// SIMATIC S7-200 project (STEP 7-Micro/WIN), CPU 226 REL 01.23

SYMBOL_TABLE analog & its vd
oil_pipe_temp0   AIW0     // oil pipe temperature channel
oil_tank_temp0   AIW2     // oil tank temperature channel
motor_draft_temp0 AIW4     // motor draft temperature channel
motor_coil1_temp0 AIW6     // motor coil 1 temperature channel
motor_coil2_temp0 AIW8     // motor coil 2 temperature channel
motor_coil3_temp0 AIW10    // motor coil 3 temperature channel
fou_out_temp0    AIW12    // fourth stage out temperature channel
thi_out_temp0    AIW14    // third stage out temperature channel
sec_out_temp0    AIW16    // second stage out temperature channel
fir_out_temp0    AIW18    // first stage out temperature channel
oil_pre0         AIW20    // oil pressure channel
delivery_pre0    AIW22    // delivery pressure channel
fou_out_pre0     AIW24    // 4th stage  out pressure channel
thi_out_pre0     AIW26    // 3rd stage  out pressure channel
sec_out_pre0     AIW28    // 2nd stage  out pressure channel
fir_out_pre0     AIW30    // 1st stage  out pressure channel
fir_in_pre0      AIW32    // 1st stage  in pressure channel
oil_pipe_temp1   VD200    // oil pipe temperature value
oil_tank_temp1   VD204    // oil tank temperature value
motor_draft_temp1 VD208    // motor draft temperature value
motor_coil3_temp1 VD212    // motor coil 1 temperature value
motor_coil2_temp1 VD216    // motor coil 2 temperature value
motor_coil1_temp1 VD220    // motor coil 3 temperature value
fou_out_temp1    VD224    // fourth stage out temperature value
thi_out_temp1    VD228    // third stage out temperature value
sec_out_temp1    VD232    // second stage out temperature value
fir_out_temp1    VD236    // first stage out temperature value
oil_pre1         VD240    // oil pressure value
delivery_pre1    VD244    // delivery pressure value
fou_out_pre1     VD248    // 4th stage  out pressure value
thi_out_pre1     VD252    // 3rd stage  out pressure value
sec_out_pre1     VD256    // 2nd stage  out pressure value
fir_out_pre1     VD260    // 1st stage  out pressure value
fir_in_pre1      VD264    // 1st stage  in pressure value
END_SYMBOL_TABLE

SYMBOL_TABLE define_m
fou_out_p_hi_p_m M10.0
oil_p_low_p_m    M10.1
fir_o_t_hi_p_m   M10.2
sec_o_t_hi_p_m   M10.3
thi_o_t_hi_p_m   M10.4
fou_o_t_hi_p_m   M10.5
fir_coil_t_hi_p_m M10.6
sec_coil_t_hi_p_m M10.7
thi_coil_t_hi_p_m M11.0
draft_t_hi_p_m   M11.1
oil_t_hi_p_m     M11.2
fir_in_p_low_p_m M11.3
fir_in_p_hi_p_m  M11.4
delivery_p_hi_p_m M11.5
fou_o_p_hi_a_m   M14.0
oil_p_low_a_m    M14.1
fir_o_t_hi_a_m   M14.2
sec_o_t_hi_a_m   M14.3
thi_o_t_hi_a_m   M14.4
fou_o_t_hi_a_m   M14.5
fir_coil_t_hi_a_m M14.6
sec_coil_t_hi_a_m M14.7
thi_coil_t_hi_a_m M15.0
draft_t_hi_a_m   M15.1
oil_t_hi_a_m     M15.2
fir_in_p_low_a_m M15.3
fir_in_p_hi_a_m  M15.4
delivery_p_hi_a_m M15.5
oil_start_heat_m M15.6
oil_stop_heat_m  M15.7
sec_pre_high_m   M16.0
thi_pre_high_m   M16.1
fou_pre_high_m   M16.2
a_cooling_fan    M19.0
a_aid_pump       M19.1
a_infuse_pump    M19.2
a_water_pump     M19.3
a_main_motor     M19.5
m_main_start     M25.0
m_main_stop      M25.1
m_cooling_fan    M25.2
m_venting_fan    M25.3
m_infuse_pump    M25.4
m_oil_heater     M25.5
m_oil_pump       M25.6
m_water_pump     M25.7
m_fir_vavle      M26.0
m_sec_vavle      M26.1
m_thi_vavle      M26.2
m_fou_vavle      M26.3
a_pro_unlock     M7.0
fou_o_p_hi_unlock M7.1
oil_p_low_unlock M7.2
fir_o_t_hi_unlock M7.3
sec_o_t_hi_unlock M7.4
thi_o_t_hi_unlock M7.5
fou_o_t_hi_unlock M7.6
fir_coil_t_hi_unlock M7.7
sec_coil_t_hi_unlock M8.0
thi_coil_t_hi_unlock M8.1
draft_t_hi_unlock M8.2
oil_t_hi_unlock  M8.3
fir_in_p_low_unlock M8.4
fir_in_p_hi_unlock M8.5
delivery_p_hi_unlock M8.6
END_SYMBOL_TABLE

SYMBOL_TABLE pro & ala setting
fou_o_p_hi_p_s   VD300    // 4th stage out pressure high protect
oil_p_low_p_s    VD304    // oilt pressure low protect
fir_o_t_hi_p_s   VD308    // 1st stage out temperature high protect
sec_o_t_hi_p_s   VD312    // 2nd stage out temperature high protect
thi_o_t_hi_p_s   VD316    // 3rd stage out temperature high protect
fou_o_t_hi_p_s   VD320    // 4th stage out temperature high protect
fir_coil_t_hi_p_s VD324    // 1st coil temperature high protect
sec_coil_t_hi_p_s VD328    // 2nd coil temperature high protect
thi_coil_t_hi_p_s VD332    // 3rd coil out temperature high protect
draft_t_hi_p_s   VD336    // draft temperature high protect
oil_t_hi_p_s     VD340    // oil temperature high protect
fir_in_p_low_p_s VD344    // 1st stage in pressure low protect
fir_in_p_hi_p_s  VD348    // 1st stage in pressure high protect
delivery_p_hi_p_s VD352    // delivery pressure high protect
fou_o_p_hi_a_s   VD400    // 4th stage out pressure high alarm
oil_p_low_a_s    VD404    // oilt pressure low alarm
fir_o_t_hi_a_s   VD408    // 1st stage out temperature high alarm
sec_o_t_hi_a_s   VD412    // 2nd stage out temperature high alarm
thi_o_t_hi_a_s   VD416    // 3rd stage out temperature high alarm
fou_o_t_hi_a_s   VD420    // 4th stage out temperature high alarm
fir_coil_t_hi_a_s VD424    // 1st coil temperature high alarm
sec_coil_t_hi_a_s VD428    // 2nd coil temperature high alarm
thi_coil_t_hi_a_s VD432    // 3rd coil out temperature high alarm
draft_t_hi_a_s   VD436    // draft temperature high alarm
oil_t_hi_a_s     VD440    // oil temperature high alarm
fir_in_p_low_a_s VD444    // 1st stage in pressure low alarm
fir_in_p_hi_a_s  VD448    // 1st stage in pressure high alarm
delivery_p_hi_a_s VD452    // delivery pressure high alarm
oil_start_heat_s VD456    // temperature that oil start to heat
oil_stop_heat_s  VD460    // temperature that oil stop to heat
sec_pre_hi_s     VD464    // second stage out  pressure high alarm
thi_pre_hi_s     VD468    // third stage out  pressure high alarm
fou_pre_hi_s     VD472    // fourth stage out  pressure high alarm
invalid_time     VW490    // unvalid running time
fan_stop_time    VW492    // time when relay to stop fan
next_start_time  VW494    // interval when run again
test_oil_time    VW496    // time when relay to test oil pressure
fir_in_p_test_time VW498    // time to relay to test first stage input pressure
stop_aid_pump_time VW500    // time relay to stop the aid oil pump when main motor start
vavle_relay_time VW502    // time relay to open vavle  when main motor start
interval_time    VW504    // when start automatically ,the interval to start step by step
main_relay_time  VW506    // after all aid equipment running,to start main motor time
relay_stop_water VW508    // when stop system ,relay time to stop water pump
relay_stop_oil   VW510    // when stop system ,relay time to stop oil pump
relay_to_test_fir_pre VW512    // when 3# vavle is open  ,relay time to test inlet pressure
END_SYMBOL_TABLE

SYMBOL_TABLE i/o
main_motor_run   I0.0
main_motor_fault I0.1
cooling_fan_run  I0.2
cooling_fan_fault I0.3
vent_fan_run     I0.4
vent_fan_fault   I0.5
infuse_oil_pump_run I0.6
infuse_oil_pump_fault I0.7
heater_run       I1.0
heater_fault     I1.1
fir_vavle_open   I1.2
sec_vavle_open   I1.3
thi_vavle_open   I1.4
esd              I1.5
local_remote     I1.6
automatic        I1.7
manu             I2.0
gas_leakage      I2.1
test             I2.2
confirm          I2.3
reset            I2.4
start_button     I2.5
stop_button      I2.6
spare            I2.7
main_motor_start Q0.0
main_motor_stop  Q0.1
cooling_fan_st   Q0.2
venting_fan_st   Q0.3
infuse_oil_pump_st Q0.4
oil_heater_st    Q0.5
oil_pump_st      Q0.6
water_pump_st    Q0.7
fir_vavle_st     Q1.0
sec_vavle_st     Q1.1
thi_vavle_st     Q1.2
fou_vavle_st     Q1.3
spare_q_2        Q1.4
est_output       Q1.5
permit_indicator Q1.6
alarm_out        Q1.7
END_SYMBOL_TABLE

ORGANIZATION_BLOCK MAIN:OB1
TITLE=“CNG加气站控制程序”。
// 
// 系统中，四级出口压力超过四级出口压力高保护设定值且四级出口压力高保护解除标志  未置位时，必须触发 四级出口压力高保护标志，以防止压缩机因压力过高受损；
// 同样，当 油压低于 油压低保护设定值且主电机运行 时，必须触发 油压低保护标志，确保润滑系统正常。
// 
// 自动控制 模块按照预定顺序启动设备：首先激活 冷却风扇自动控制标志，通过 启动延时定时器 延时后启动 辅助泵自动控制标志，依次启动 输油泵自动控制标志、水泵自动控制标志，最后启动 主电机自动控制标志，每步之间必须有延时以确保设备稳定运行。
// 输出控制 根据逻辑驱动实际设备，主电机启动输出 仅在 主电机自动控制标志或手动启动信号有效时才能置位，而 报警输出 必须在系统异常（如 四级出口压力高保护标志 触发时）或紧急停机触发时激活，确保操作员及时响应。
// 
// 报警逻辑监测异常情况，当 四级出口压力超过 四级出口压力高报警设定值 时，必须触发 四级出口压力高报警标志，提醒维护人员检查系统。
// 此外，恢复出厂设置功能允许将 四级出口压力高保护设定值等参数重置为默认值（25.0）。
BEGIN
Network 1 // 网络标题
// 网络注释
LD     SM0.0
LPS
CALL   analog:SBR0
AN     a_pro_unlock:M7.0
CALL   protect:SBR1
LRD
CALL   alarm:SBR6
LPP
AW=    0, MW10
=      M28.0
Network 2 // 网络标题
// 网络注释
LDN    automatic:I1.7
AN     manu:I2.0
=      M28.5
Network 3
LD     reset:I2.4
MOVW   0, MW10
MOVW   0, MW14
MOVW   0, MW16
Network 4
LDN    main_motor_fault:I0.1
AN     cooling_fan_fault:I0.3
AN     vent_fan_fault:I0.5
AN     infuse_oil_pump_fault:I0.7
AN     heater_fault:I1.1
=      M28.1
Network 5
LD     M28.0
A      M28.1
AN     esd:I1.5
A      automatic:I1.7
CALL   auto:SBR2
Network 6
LDN    M28.0
ON     M28.1
O      esd:I1.5
ON     automatic:I1.7
MOVW   0, MW19
=      alarm_out:Q1.7
Network 7
LDN    manu:I2.0
MOVW   0, MW25
Network 8
LD     confirm:I2.3
A      reset:I2.4
TON    T40, 100
Network 9
LD     T40
CALL   recovery:SBR7
Network 10
LD     automatic:I1.7
O      manu:I2.0
A      M28.0
A      M28.1
AN     esd:I1.5
AN     M0.0
CALL   out:SBR4
Network 11 // 网络标题
// 网络注释
LD     esd:I1.5
=      est_output:Q1.5
END_ORGANIZATION_BLOCK

SUBROUTINE_BLOCK analog:SBR0
TITLE=子程序注释
BEGIN
Network 1
LD     SM0.0
CALL   Temperature:SBR11, oil_pipe_temp0:AIW0, oil_pipe_temp1:VD200
CALL   Temperature:SBR11, oil_tank_temp0:AIW2, oil_tank_temp1:VD204
CALL   Temperature:SBR11, motor_draft_temp0:AIW4, motor_draft_temp1:VD208
CALL   Temperature:SBR11, motor_coil3_temp0:AIW10, motor_coil3_temp1:VD212
CALL   Temperature:SBR11, motor_coil2_temp0:AIW8, motor_coil2_temp1:VD216
CALL   Temperature:SBR11, motor_coil1_temp0:AIW6, motor_coil1_temp1:VD220
CALL   Temperature:SBR11, fou_out_temp0:AIW12, fou_out_temp1:VD224
CALL   Temperature:SBR11, thi_out_temp0:AIW14, thi_out_temp1:VD228
CALL   Temperature:SBR11, sec_out_temp0:AIW16, sec_out_temp1:VD232
CALL   Temperature:SBR11, fir_out_temp0:AIW18, fir_out_temp1:VD236
Network 2 // 网络标题
// 网络注释
LD     SM0.0
CALL   Pressure:SBR12, oil_pre0:AIW20, 1.6, oil_pre1:VD240
CALL   Pressure:SBR12, delivery_pre0:AIW22, 40.0, delivery_pre1:VD244
CALL   Pressure:SBR12, fou_out_pre0:AIW24, 40.0, fou_out_pre1:VD248
CALL   Pressure:SBR12, thi_out_pre0:AIW26, 25.0, thi_out_pre1:VD252
CALL   Pressure:SBR12, sec_out_pre0:AIW28, 10.0, sec_out_pre1:VD256
CALL   Pressure:SBR12, fir_out_pre0:AIW30, 4.0, fir_out_pre1:VD260
CALL   Pressure:SBR12, fir_in_pre0:AIW32, 1.6, fir_in_pre1:VD264
END_SUBROUTINE_BLOCK

SUBROUTINE_BLOCK protect:SBR1
TITLE=
BEGIN
Network 1
LDR>=  fou_out_pre1:VD248, fou_o_p_hi_p_s:VD300
O      fou_out_p_hi_p_m:M10.0
AN     fou_o_p_hi_unlock:M7.1
=      fou_out_p_hi_p_m:M10.0
Network 2
LD     oil_pump_st:Q0.6
TON    T38, test_oil_time:VW496
Network 3
LD     T38
O      M19.6
AR>=   oil_p_low_p_s:VD304, oil_pre1:VD240
O      oil_p_low_p_m:M10.1
AN     oil_p_low_unlock:M7.2
=      oil_p_low_p_m:M10.1
Network 4
LDR>=  fir_out_temp1:VD236, fir_o_t_hi_p_s:VD308
O      fir_o_t_hi_p_m:M10.2
AN     fir_o_t_hi_unlock:M7.3
=      fir_o_t_hi_p_m:M10.2
Network 5
LDR>=  sec_out_temp1:VD232, sec_o_t_hi_p_s:VD312
O      sec_o_t_hi_p_m:M10.3
AN     sec_o_t_hi_unlock:M7.4
=      sec_o_t_hi_p_m:M10.3
Network 6
LDR>=  thi_out_temp1:VD228, thi_o_t_hi_p_s:VD316
O      thi_o_t_hi_p_m:M10.4
AN     thi_o_t_hi_unlock:M7.5
=      thi_o_t_hi_p_m:M10.4
Network 7
LDR>=  fou_out_temp1:VD224, fou_o_t_hi_p_s:VD320
O      fou_o_t_hi_p_m:M10.5
AN     fou_o_t_hi_unlock:M7.6
=      fou_o_t_hi_p_m:M10.5
Network 8
LDR>=  motor_coil1_temp1:VD220, fir_coil_t_hi_p_s:VD324
O      fir_coil_t_hi_p_m:M10.6
AN     fir_coil_t_hi_unlock:M7.7
=      fir_coil_t_hi_p_m:M10.6
Network 9
LDR>=  motor_coil2_temp1:VD216, sec_coil_t_hi_p_s:VD328
O      sec_coil_t_hi_p_m:M10.7
AN     sec_coil_t_hi_unlock:M8.0
=      sec_coil_t_hi_p_m:M10.7
Network 10
LDR>=  motor_coil3_temp1:VD212, thi_coil_t_hi_p_s:VD332
O      thi_coil_t_hi_p_m:M11.0
AN     thi_coil_t_hi_unlock:M8.1
=      thi_coil_t_hi_p_m:M11.0
Network 11
LDR>=  motor_draft_temp1:VD208, draft_t_hi_p_s:VD336
O      draft_t_hi_p_m:M11.1
AN     draft_t_hi_unlock:M8.2
=      draft_t_hi_p_m:M11.1
Network 12
LDR>=  oil_pipe_temp1:VD200, oil_t_hi_p_s:VD340
O      oil_t_hi_p_m:M11.2
AN     oil_t_hi_unlock:M8.3
=      oil_t_hi_p_m:M11.2
Network 13
LD     thi_vavle_st:Q1.2
TON    T39, relay_to_test_fir_pre:VW512
Network 14
LD     T39
AR>=   fir_in_p_low_p_s:VD344, fir_in_pre1:VD264
O      fir_in_p_low_p_m:M11.3
AN     fir_in_p_low_unlock:M8.4
=      fir_in_p_low_p_m:M11.3
Network 15
LD     T39
AR>=   fir_in_pre1:VD264, fir_in_p_hi_p_s:VD348
O      fir_in_p_hi_p_m:M11.4
AN     fir_in_p_hi_unlock:M8.5
=      fir_in_p_hi_p_m:M11.4
Network 16
LDR>=  delivery_pre1:VD244, delivery_p_hi_p_s:VD352
O      delivery_p_hi_p_m:M11.5
AN     delivery_p_hi_unlock:M8.6
=      delivery_p_hi_p_m:M11.5
END_SUBROUTINE_BLOCK

SUBROUTINE_BLOCK auto:SBR2
TITLE=
BEGIN
Network 1
LD     start_button:I2.5
O      a_cooling_fan:M19.0
AN     T23
=      a_cooling_fan:M19.0
TONR   T10, interval_time:VW504
Network 2
LD     T10
O      a_aid_pump:M19.1
AN     T15
=      a_aid_pump:M19.1
TONR   T11, interval_time:VW504
Network 3
LD     T11
O      a_infuse_pump:M19.2
AN     T22
=      a_infuse_pump:M19.2
TONR   T12, interval_time:VW504
Network 4
LD     T12
O      a_water_pump:M19.3
AN     T21
=      a_water_pump:M19.3
TONR   T13, interval_time:VW504
Network 5
LD     T13
O      M19.4
AN     a_main_motor:M19.5
=      M19.4
TONR   T14, main_relay_time:VW506
Network 6
LD     T14
O      a_main_motor:M19.5
AN     M19.6
=      a_main_motor:M19.5
TONR   T15, stop_aid_pump_time:VW500
Network 7
LD     T14
O      M19.6
AN     M19.7
=      M19.6
TONR   T16, vavle_relay_time:VW502
Network 8
LDR>=  delivery_pre1:VD244, delivery_p_hi_p_s:VD352
TONR   T19, 20
Network 9
LD     stop_button:I2.6
O      T19
A      M19.6
O      M19.7
AN     M20.0
=      M19.7
TONR   T20, invalid_time:VW490
Network 10
LD     T20
O      M20.0
AN     M20.1
=      M20.0
TONR   T21, relay_stop_water:VW508
Network 11
LD     T21
O      M20.1
AN     M20.2
=      M20.1
TONR   T22, relay_stop_oil:VW510
Network 12
LD     T22
O      M20.2
AN     T23
=      M20.2
TONR   T23, fan_stop_time:VW492
END_SUBROUTINE_BLOCK

SUBROUTINE_BLOCK sense:SBR3
TITLE=子程序注释
BEGIN
Network 1 //  网络标题
//  网络注解
LD     SM0.4
EU
INCD   VD1000
Network 2
LDD>=  VD1000, 36000
O      M0.0
AN     T105
=      M0.0
Network 3
LD     esd:I1.5
A      reset:I2.4
A      confirm:I2.3
A      manu:I2.0
TON    T105, 150
Network 4
LD     T105
MOVD   0, VD1000
Network 5 // 网络标题
// 网络注释
END_SUBROUTINE_BLOCK

SUBROUTINE_BLOCK out:SBR4
TITLE=子程序注释
BEGIN
Network 1 // 网络标题
// 网络注释
LD     m_main_start:M25.0
TON    T40, 30
Network 2 // 网络标题
// 网络注释
LD     T40
R      m_main_start:M25.0, 1
Network 3 // 网络标题
// 网络注释
LD     m_main_stop:M25.1
TON    T41, 30
Network 4 // 网络标题
// 网络注释
LD     T41
R      m_main_stop:M25.1, 1
Network 5 // 网络标题
// 网络注释
LD     a_main_motor:M19.5
O      m_main_start:M25.0
=      main_motor_start:Q0.0
Network 6 // 网络标题
// 网络注释
LD     M20.0
O      m_main_stop:M25.1
=      main_motor_stop:Q0.1
Network 7 // 网络标题
// 网络注释
LD     a_cooling_fan:M19.0
O      m_cooling_fan:M25.2
=      cooling_fan_st:Q0.2
Network 8 // 网络标题
// 网络注释
LD     gas_leakage:I2.1
ED
O      M3.1
LPS
AN     T43
=      M3.1
LPP
TON    T43, 500
Network 9 // 网络标题
// 网络注释
LD     gas_leakage:I2.1
O      M3.1
O      m_venting_fan:M25.3
=      venting_fan_st:Q0.3
Network 10 // 网络标题
// 网络注释
LD     a_infuse_pump:M19.2
O      m_infuse_pump:M25.4
=      infuse_oil_pump_st:Q0.4
Network 11 // 网络标题
// 网络注释
LD     a_aid_pump:M19.1
O      m_oil_heater:M25.5
=      oil_heater_st:Q0.5
Network 12 // 网络标题
// 网络注释
LD     a_infuse_pump:M19.2
O      m_oil_pump:M25.6
=      oil_pump_st:Q0.6
Network 13 // 网络标题
// 网络注释
LD     a_water_pump:M19.3
O      m_water_pump:M25.7
=      water_pump_st:Q0.7
Network 14 // 网络标题
// 网络注释
LD     a_cooling_fan:M19.0
O      m_sec_vavle:M26.1
=      fir_vavle_st:Q1.0
Network 15 // 网络标题
// 网络注释
LD     a_cooling_fan:M19.0
O      m_thi_vavle:M26.2
=      sec_vavle_st:Q1.1
Network 16 // 网络标题
// 网络注释
LD     a_cooling_fan:M19.0
O      m_fou_vavle:M26.3
=      thi_vavle_st:Q1.2
Network 17 // 网络标题
// 网络注释
LD     SM0.0
=      permit_indicator:Q1.6
END_SUBROUTINE_BLOCK

SUBROUTINE_BLOCK interlock:SBR5
TITLE=
BEGIN
Network 1
LD     oil_p_low_p_m:M10.1
AN     M13.1
LD     fir_coil_t_hi_p_m:M10.6
AN     M13.4
OLD
LD     thi_coil_t_hi_p_m:M11.0
AN     M13.5
OLD
LD     oil_t_hi_p_m:M11.2
AN     M13.6
OLD
LD     fir_in_p_hi_p_m:M11.4
AN     M13.7
OLD
LD     M11.6
AN     fou_o_p_hi_a_m:M14.0
OLD
LD     M12.0
AN     oil_p_low_a_m:M14.1
OLD
LD     M12.2
AN     fir_o_t_hi_a_m:M14.2
OLD
LD     M12.4
AN     sec_o_t_hi_a_m:M14.3
OLD
LD     M12.6
AN     thi_o_t_hi_a_m:M14.4
OLD
LD     fir_coil_t_hi_a_m:M14.6
AN     reset:I2.4
OLD
AN     fou_o_t_hi_a_m:M14.5
=      fir_coil_t_hi_a_m:M14.6
END_SUBROUTINE_BLOCK

SUBROUTINE_BLOCK alarm:SBR6
TITLE=
BEGIN
Network 1
LDR>=  fou_out_pre1:VD248, fou_o_p_hi_a_s:VD400
O      fou_o_p_hi_a_m:M14.0
=      fou_o_p_hi_a_m:M14.0
Network 2
LD     T38
O      M19.6
AR>=   oil_p_low_a_s:VD404, oil_pre1:VD240
O      oil_p_low_a_m:M14.1
=      oil_p_low_a_m:M14.1
Network 3
LDR>=  fir_out_temp1:VD236, fir_o_t_hi_a_s:VD408
O      fir_o_t_hi_a_m:M14.2
=      fir_o_t_hi_a_m:M14.2
Network 4
LDR>=  sec_out_temp1:VD232, sec_o_t_hi_a_s:VD412
O      sec_o_t_hi_a_m:M14.3
=      sec_o_t_hi_a_m:M14.3
Network 5
LDR>=  thi_out_temp1:VD228, thi_o_t_hi_a_s:VD416
O      thi_o_t_hi_a_m:M14.4
=      thi_o_t_hi_a_m:M14.4
Network 6
LDR>=  fou_out_temp1:VD224, fou_o_t_hi_a_s:VD420
O      fou_o_t_hi_a_m:M14.5
=      fou_o_t_hi_a_m:M14.5
Network 7
LDR>=  motor_coil1_temp1:VD220, fir_coil_t_hi_a_s:VD424
O      fir_coil_t_hi_a_m:M14.6
=      fir_coil_t_hi_a_m:M14.6
Network 8
LDR>=  motor_coil2_temp1:VD216, sec_coil_t_hi_a_s:VD428
O      sec_coil_t_hi_a_m:M14.7
=      sec_coil_t_hi_a_m:M14.7
Network 9
LDR>=  motor_coil3_temp1:VD212, thi_coil_t_hi_a_s:VD432
O      thi_coil_t_hi_a_m:M15.0
=      thi_coil_t_hi_a_m:M15.0
Network 10
LDR>=  motor_draft_temp1:VD208, draft_t_hi_a_s:VD436
O      draft_t_hi_a_m:M15.1
=      draft_t_hi_a_m:M15.1
Network 11
LDR>=  oil_pipe_temp1:VD200, oil_t_hi_a_s:VD440
O      oil_t_hi_a_m:M15.2
=      oil_t_hi_a_m:M15.2
Network 12
LD     T39
AR>=   fir_in_p_low_a_s:VD444, fir_in_pre1:VD264
O      fir_in_p_low_a_m:M15.3
=      fir_in_p_low_a_m:M15.3
Network 13
LD     T39
AR>=   fir_in_pre1:VD264, fir_in_p_hi_a_s:VD448
O      fir_in_p_hi_a_m:M15.4
=      fir_in_p_hi_a_m:M15.4
Network 14
LDR>=  delivery_pre1:VD244, delivery_p_hi_a_s:VD452
O      delivery_p_hi_a_m:M15.5
=      delivery_p_hi_a_m:M15.5
Network 15
LDR>=  oil_start_heat_s:VD456, oil_tank_temp1:VD204
O      oil_start_heat_m:M15.6
=      oil_start_heat_m:M15.6
Network 16
LDR>=  oil_tank_temp1:VD204, oil_stop_heat_s:VD460
O      oil_stop_heat_m:M15.7
=      oil_stop_heat_m:M15.7
Network 17
LDR>=  sec_out_pre1:VD256, sec_pre_hi_s:VD464
O      sec_pre_high_m:M16.0
=      sec_pre_high_m:M16.0
Network 18
LDR>=  thi_out_pre1:VD252, thi_pre_hi_s:VD468
O      thi_pre_high_m:M16.1
=      thi_pre_high_m:M16.1
Network 19
LDR>=  fou_out_pre1:VD248, fou_pre_hi_s:VD472
O      fou_pre_high_m:M16.2
=      fou_pre_high_m:M16.2
END_SUBROUTINE_BLOCK

SUBROUTINE_BLOCK recovery:SBR7
TITLE=
BEGIN
Network 1
//  set protecting parameters will be recovered by the factory setting datas
LD     SM0.0
LPS
MOVR   25.0, fou_o_p_hi_p_s:VD300
AENO
MOVR   0.15, oil_p_low_p_s:VD304
LRD
MOVR   150.0, fir_o_t_hi_p_s:VD308
AENO
MOVR   150.0, sec_o_t_hi_p_s:VD312
LRD
MOVR   150.0, thi_o_t_hi_p_s:VD316
AENO
MOVR   150.0, fou_o_t_hi_p_s:VD320
LRD
MOVR   95.0, fir_coil_t_hi_p_s:VD324
AENO
MOVR   95.0, sec_coil_t_hi_p_s:VD328
LRD
MOVR   95.0, thi_coil_t_hi_p_s:VD332
AENO
MOVR   60.0, draft_t_hi_p_s:VD336
LRD
MOVR   55.0, oil_t_hi_p_s:VD340
AENO
MOVR   4.5, fir_in_p_low_p_s:VD344
LPP
MOVR   8.0, fir_in_p_hi_p_s:VD348
AENO
MOVR   25.0, delivery_p_hi_p_s:VD352
Network 2
//  set alarm parameters will be recovered by the factory setting datas
LD     SM0.0
LPS
MOVR   25.0, fou_o_p_hi_a_s:VD400
AENO
MOVR   0.15, oil_p_low_a_s:VD404
LRD
MOVR   150.0, fir_o_t_hi_a_s:VD408
AENO
MOVR   150.0, sec_o_t_hi_a_s:VD412
LRD
MOVR   150.0, thi_o_t_hi_a_s:VD416
AENO
MOVR   150.0, fou_o_t_hi_a_s:VD420
LRD
MOVR   95.0, fir_coil_t_hi_a_s:VD424
AENO
MOVR   95.0, sec_coil_t_hi_a_s:VD428
LRD
MOVR   95.0, thi_coil_t_hi_a_s:VD432
AENO
MOVR   60.0, draft_t_hi_a_s:VD436
LRD
MOVR   55.0, oil_t_hi_a_s:VD440
AENO
MOVR   4.5, fir_in_p_low_a_s:VD444
LRD
MOVR   8.0, fir_in_p_hi_a_s:VD448
AENO
MOVR   25.0, delivery_p_hi_a_s:VD452
LRD
MOVR   5.0, oil_start_heat_s:VD456
AENO
MOVR   15.0, oil_stop_heat_s:VD460
LRD
MOVR   2.5, sec_pre_hi_s:VD464
AENO
MOVR   7.6, thi_pre_hi_s:VD468
LPP
MOVR   14.9, fou_pre_hi_s:VD472
Network 3
//  set alarm parameters will be recovered by the factory setting datas
LD     SM0.0
LPS
MOVW   100, invalid_time:VW490
AENO
MOVW   100, fan_stop_time:VW492
LRD
MOVW   100, next_start_time:VW494
AENO
MOVW   100, test_oil_time:VW496
LRD
MOVW   100, fir_in_p_test_time:VW498
AENO
MOVW   100, stop_aid_pump_time:VW500
LRD
MOVW   100, vavle_relay_time:VW502
AENO
MOVW   100, interval_time:VW504
LPP
MOVW   100, main_relay_time:VW506
AENO
MOVW   100, relay_stop_water:VW508
END_SUBROUTINE_BLOCK
